// TIA Portal V15.1 export
// export: Created 2019-08-08T13:49:45.9027601Z, ExportSetting None, DisplayName Totally Integrated Automation Portal, DisplayVersion V15.1, DisplayName TIA Portal Openness, DisplayVersion V15.1, DisplayName STEP 7 Professional, DisplayVersion V15.1, DisplayName STEP 7 Safety, DisplayVersion V15.1, DisplayName WinCC Advanced, DisplayVersion V15.1
TYPE "typeSkillStateMachineMapping"
   STRUCT
      StateMachine : Struct
         CurrentState_Id : OPC_UA_NodeId;
         LastTransition_Id : OPC_UA_NodeId;
         AvailableStates_NodeIds : Array[0..2] of OPC_UA_NodeId;
         AvailableStates_Names : Array[0..2] of String;
         AvailableStates_Numbers : Array[0..2] of Byte;
         AvailableTransitions_NodeIds : Array[0..2] of OPC_UA_NodeId;
         AvailableTransitions_Names : Array[0..2] of String;
         AvailableTransitions_Numbers : Array[0..2] of Byte;
      END_STRUCT;
      ClearedStateMachine : Struct
         CurrentState_Id : OPC_UA_NodeId;
         LastTransition_Id : OPC_UA_NodeId;
         AvailableStates_NodeIds : Array[0..3] of OPC_UA_NodeId;
         AvailableStates_Names : Array[0..3] of String;
         AvailableStates_Numbers : Array[0..3] of Byte;
         AvailableTransitions_NodeIds : Array[0..3] of OPC_UA_NodeId;
         AvailableTransitions_Names : Array[0..3] of String;
         AvailableTransitions_Numbers : Array[0..3] of Byte;
      END_STRUCT;
      RunningStateMachine : Struct
         CurrentState_Id : OPC_UA_NodeId;
         LastTransition_Id : OPC_UA_NodeId;
         AvailableStates_NodeIds : Array[0..5] of OPC_UA_NodeId;
         AvailableStates_Names : Array[0..5] of String;
         AvailableStates_Numbers : Array[0..5] of Byte;
         AvailableTransitions_NodeIds : Array[0..6] of OPC_UA_NodeId;
         AvailableTransitions_Names : Array[0..6] of String;
         AvailableTransitions_Numbers : Array[0..6] of Byte;
      END_STRUCT;
      IdleStateMachine : Struct
         CurrentState_Id : OPC_UA_NodeId;
         LastTransition_Id : OPC_UA_NodeId;
         AvailableStates_NodeIds : Array[0..1] of OPC_UA_NodeId;
         AvailableStates_Names : Array[0..1] of String;
         AvailableStates_Numbers : Array[0..1] of Byte;
         AvailableTransitions_NodeIds : Array[0..0] of OPC_UA_NodeId;
         AvailableTransitions_Names : Array[0..0] of String;
         AvailableTransitions_Numbers : Array[0..0] of Byte;
      END_STRUCT;
      HoldStateMachine : Struct
         CurrentState_Id : OPC_UA_NodeId;
         LastTransition_Id : OPC_UA_NodeId;
         AvailableStates_NodeIds : Array[0..2] of OPC_UA_NodeId;
         AvailableStates_Names : Array[0..2] of String;
         AvailableStates_Numbers : Array[0..2] of Byte;
         AvailableTransitions_NodeIds : Array[0..1] of OPC_UA_NodeId;
         AvailableTransitions_Names : Array[0..1] of String;
         AvailableTransitions_Numbers : Array[0..1] of Byte;
      END_STRUCT;
      ResettingStateMachine : Struct
         CurrentState_Id : OPC_UA_NodeId;
         LastTransition_Id : OPC_UA_NodeId;
         AvailableStates_NodeIds : Array[0..2] of OPC_UA_NodeId;
         AvailableStates_Names : Array[0..2] of String;
         AvailableStates_Numbers : Array[0..2] of Byte;
         AvailableTransitions_NodeIds : Array[0..2] of OPC_UA_NodeId;
         AvailableTransitions_Names : Array[0..2] of String;
         AvailableTransitions_Numbers : Array[0..2] of Byte;
      END_STRUCT;
      ExecuteStateMachine : Struct
         CurrentState_Id : OPC_UA_NodeId;
         LastTransition_Id : OPC_UA_NodeId;
         AvailableStates_NodeIds : Array[0..1] of OPC_UA_NodeId;
         AvailableStates_Names : Array[0..1] of String;
         AvailableStates_Numbers : Array[0..1] of Byte;
         AvailableTransitions_NodeIds : Array[0..1] of OPC_UA_NodeId;
         AvailableTransitions_Names : Array[0..1] of String;
         AvailableTransitions_Numbers : Array[0..1] of Byte;
      END_STRUCT;
   END_STRUCT;
   // StateMachine.AvailableStates_NodeIds[0].Identifier := WSTRING#'71';
   // StateMachine.AvailableStates_NodeIds[1].Identifier := WSTRING#'61';
   // StateMachine.AvailableStates_NodeIds[2].Identifier := WSTRING#'62';
   // StateMachine.AvailableStates_Names[0] := 'Cleared';
   // StateMachine.AvailableStates_Names[1] := 'Aborting';
   // StateMachine.AvailableStates_Names[2] := 'Aborted';
   // StateMachine.AvailableStates_Numbers[0] := 1;
   // StateMachine.AvailableStates_Numbers[1] := 2;
   // StateMachine.AvailableStates_Numbers[2] := 3;
   // StateMachine.AvailableTransitions_NodeIds[0].Identifier := WSTRING#'1007';
   // StateMachine.AvailableTransitions_NodeIds[1].Identifier := WSTRING#'1008';
   // StateMachine.AvailableTransitions_NodeIds[2].Identifier := WSTRING#'66';
   // StateMachine.AvailableTransitions_Names[0] := 'ClearedToAborting';
   // StateMachine.AvailableTransitions_Names[1] := 'AbortedToCleared';
   // StateMachine.AvailableTransitions_Names[2] := 'AbortingToAborted';
   // StateMachine.AvailableTransitions_Numbers[0] := 1;
   // StateMachine.AvailableTransitions_Numbers[1] := 2;
   // StateMachine.AvailableTransitions_Numbers[2] := 3;
   // ClearedStateMachine.AvailableStates_NodeIds[0].Identifier := WSTRING#'55';
   // ClearedStateMachine.AvailableStates_NodeIds[1].Identifier := WSTRING#'53';
   // ClearedStateMachine.AvailableStates_NodeIds[2].Identifier := WSTRING#'75';
   // ClearedStateMachine.AvailableStates_NodeIds[3].Identifier := WSTRING#'54';
   // ClearedStateMachine.AvailableStates_Names[0] := 'Clearing';
   // ClearedStateMachine.AvailableStates_Names[1] := 'Stopped';
   // ClearedStateMachine.AvailableStates_Names[2] := 'Running';
   // ClearedStateMachine.AvailableStates_Names[3] := 'Stopping';
   // ClearedStateMachine.AvailableStates_Numbers[0] := 1;
   // ClearedStateMachine.AvailableStates_Numbers[1] := 2;
   // ClearedStateMachine.AvailableStates_Numbers[2] := 3;
   // ClearedStateMachine.AvailableStates_Numbers[3] := 4;
   // ClearedStateMachine.AvailableTransitions_NodeIds[0].Identifier := WSTRING#'58';
   // ClearedStateMachine.AvailableTransitions_NodeIds[1].Identifier := WSTRING#'1000';
   // ClearedStateMachine.AvailableTransitions_NodeIds[2].Identifier := WSTRING#'1006';
   // ClearedStateMachine.AvailableTransitions_NodeIds[3].Identifier := WSTRING#'57';
   // ClearedStateMachine.AvailableTransitions_Names[0] := 'ClearingToStopped';
   // ClearedStateMachine.AvailableTransitions_Names[1] := 'StoppedToRunning';
   // ClearedStateMachine.AvailableTransitions_Names[2] := 'RunningToStopping';
   // ClearedStateMachine.AvailableTransitions_Names[3] := 'StoppingToStopped';
   // ClearedStateMachine.AvailableTransitions_Numbers[0] := 1;
   // ClearedStateMachine.AvailableTransitions_Numbers[1] := 2;
   // ClearedStateMachine.AvailableTransitions_Numbers[2] := 3;
   // ClearedStateMachine.AvailableTransitions_Numbers[3] := 4;
   // RunningStateMachine.AvailableStates_NodeIds[0].Identifier := WSTRING#'27';
   // RunningStateMachine.AvailableStates_NodeIds[1].Identifier := WSTRING#'28';
   // RunningStateMachine.AvailableStates_NodeIds[2].Identifier := WSTRING#'36';
   // RunningStateMachine.AvailableStates_NodeIds[3].Identifier := WSTRING#'1036';
   // RunningStateMachine.AvailableStates_NodeIds[4].Identifier := WSTRING#'37';
   // RunningStateMachine.AvailableStates_NodeIds[5].Identifier := WSTRING#'38';
   // RunningStateMachine.AvailableStates_Names[0] := 'Resetting';
   // RunningStateMachine.AvailableStates_Names[1] := 'Idle';
   // RunningStateMachine.AvailableStates_Names[2] := 'Execute';
   // RunningStateMachine.AvailableStates_Names[3] := 'Hold';
   // RunningStateMachine.AvailableStates_Names[4] := 'Completing';
   // RunningStateMachine.AvailableStates_Names[5] := 'Complete';
   // RunningStateMachine.AvailableStates_Numbers[0] := 1;
   // RunningStateMachine.AvailableStates_Numbers[1] := 2;
   // RunningStateMachine.AvailableStates_Numbers[2] := 3;
   // RunningStateMachine.AvailableStates_Numbers[3] := 4;
   // RunningStateMachine.AvailableStates_Numbers[4] := 5;
   // RunningStateMachine.AvailableStates_Numbers[5] := 6;
   // RunningStateMachine.AvailableTransitions_NodeIds[0].Identifier := WSTRING#'39';
   // RunningStateMachine.AvailableTransitions_NodeIds[1].Identifier := WSTRING#'1002';
   // RunningStateMachine.AvailableTransitions_NodeIds[2].Identifier := WSTRING#'1041';
   // RunningStateMachine.AvailableTransitions_NodeIds[3].Identifier := WSTRING#'1040';
   // RunningStateMachine.AvailableTransitions_NodeIds[4].Identifier := WSTRING#'1003';
   // RunningStateMachine.AvailableTransitions_NodeIds[5].Identifier := WSTRING#'50';
   // RunningStateMachine.AvailableTransitions_NodeIds[6].Identifier := WSTRING#'1042';
   // RunningStateMachine.AvailableTransitions_Names[0] := 'ResettingToIdle';
   // RunningStateMachine.AvailableTransitions_Names[1] := 'IdleToExecute';
   // RunningStateMachine.AvailableTransitions_Names[2] := 'ExecuteToHold';
   // RunningStateMachine.AvailableTransitions_Names[3] := 'HoldToExecute';
   // RunningStateMachine.AvailableTransitions_Names[4] := 'ExecuteToCompleting';
   // RunningStateMachine.AvailableTransitions_Names[5] := 'CompletingToComplete';
   // RunningStateMachine.AvailableTransitions_Names[6] := 'CompleteToIdle';
   // RunningStateMachine.AvailableTransitions_Numbers[0] := 1;
   // RunningStateMachine.AvailableTransitions_Numbers[1] := 2;
   // RunningStateMachine.AvailableTransitions_Numbers[2] := 3;
   // RunningStateMachine.AvailableTransitions_Numbers[3] := 4;
   // RunningStateMachine.AvailableTransitions_Numbers[4] := 5;
   // RunningStateMachine.AvailableTransitions_Numbers[5] := 6;
   // RunningStateMachine.AvailableTransitions_Numbers[6] := 7;
   // IdleStateMachine.AvailableStates_NodeIds[0].Identifier := WSTRING#'1018';
   // IdleStateMachine.AvailableStates_NodeIds[1].Identifier := WSTRING#'1017';
   // IdleStateMachine.AvailableStates_Names[0] := 'InitializeSkill';
   // IdleStateMachine.AvailableStates_Names[1] := 'SkillReady';
   // IdleStateMachine.AvailableStates_Numbers[0] := 1;
   // IdleStateMachine.AvailableStates_Numbers[1] := 2;
   // IdleStateMachine.AvailableTransitions_NodeIds[0].Identifier := WSTRING#'1019';
   // IdleStateMachine.AvailableTransitions_Names[0] := 'InitializeSkillToSkillReady';
   // IdleStateMachine.AvailableTransitions_Numbers[0] := 1;
   // HoldStateMachine.AvailableStates_NodeIds[0].Identifier := WSTRING#'1020';
   // HoldStateMachine.AvailableStates_NodeIds[1].Identifier := WSTRING#'1021';
   // HoldStateMachine.AvailableStates_NodeIds[2].Identifier := WSTRING#'1022';
   // HoldStateMachine.AvailableStates_Names[0] := 'Holding';
   // HoldStateMachine.AvailableStates_Names[1] := 'Held';
   // HoldStateMachine.AvailableStates_Names[2] := 'Unholding';
   // HoldStateMachine.AvailableStates_Numbers[0] := 1;
   // HoldStateMachine.AvailableStates_Numbers[1] := 2;
   // HoldStateMachine.AvailableStates_Numbers[2] := 3;
   // HoldStateMachine.AvailableTransitions_NodeIds[0].Identifier := WSTRING#'1024';
   // HoldStateMachine.AvailableTransitions_NodeIds[1].Identifier := WSTRING#'1023';
   // HoldStateMachine.AvailableTransitions_Names[0] := 'HeldToUnholding';
   // HoldStateMachine.AvailableTransitions_Names[1] := 'HoldingToHeld';
   // HoldStateMachine.AvailableTransitions_Numbers[0] := 1;
   // HoldStateMachine.AvailableTransitions_Numbers[1] := 2;
   // ResettingStateMachine.AvailableStates_NodeIds[0].Identifier := WSTRING#'1026';
   // ResettingStateMachine.AvailableStates_NodeIds[1].Identifier := WSTRING#'1025';
   // ResettingStateMachine.AvailableStates_NodeIds[2].Identifier := WSTRING#'1027';
   // ResettingStateMachine.AvailableStates_Names[0] := 'CheckSkillComponent';
   // ResettingStateMachine.AvailableStates_Names[1] := 'InitializeSkillComponent';
   // ResettingStateMachine.AvailableStates_Names[2] := 'SkillComponentsReady';
   // ResettingStateMachine.AvailableStates_Numbers[0] := 1;
   // ResettingStateMachine.AvailableStates_Numbers[1] := 2;
   // ResettingStateMachine.AvailableStates_Numbers[2] := 3;
   // ResettingStateMachine.AvailableTransitions_NodeIds[0].Identifier := WSTRING#'1028';
   // ResettingStateMachine.AvailableTransitions_NodeIds[1].Identifier := WSTRING#'10230';
   // ResettingStateMachine.AvailableTransitions_NodeIds[2].Identifier := WSTRING#'1029';
   // ResettingStateMachine.AvailableTransitions_Names[0] := 'CheckSkillComponentToInitializeSkillComponent';
   // ResettingStateMachine.AvailableTransitions_Names[1] := 'CheckSkillComponentToSkillComponentsReady';
   // ResettingStateMachine.AvailableTransitions_Names[2] := 'InitializeSkillComponentToCheckSkillComponent';
   // ResettingStateMachine.AvailableTransitions_Numbers[0] := 1;
   // ResettingStateMachine.AvailableTransitions_Numbers[1] := 2;
   // ResettingStateMachine.AvailableTransitions_Numbers[2] := 3;
   // ExecuteStateMachine.AvailableStates_NodeIds[0].Identifier := WSTRING#'1013';
   // ExecuteStateMachine.AvailableStates_NodeIds[1].Identifier := WSTRING#'1014';
   // ExecuteStateMachine.AvailableStates_Names[0] := 'ExecuteSkill';
   // ExecuteStateMachine.AvailableStates_Names[1] := 'WaitForNextStep';
   // ExecuteStateMachine.AvailableStates_Numbers[0] := 1;
   // ExecuteStateMachine.AvailableStates_Numbers[1] := 2;
   // ExecuteStateMachine.AvailableTransitions_NodeIds[0].Identifier := WSTRING#'1015';
   // ExecuteStateMachine.AvailableTransitions_NodeIds[1].Identifier := WSTRING#'1016';
   // ExecuteStateMachine.AvailableTransitions_Names[0] := 'ExecuteSkillToWaitForNextStep';
   // ExecuteStateMachine.AvailableTransitions_Names[1] := 'WaitForNextStepToExecuteSkill';
   // ExecuteStateMachine.AvailableTransitions_Numbers[0] := 1;
   // ExecuteStateMachine.AvailableTransitions_Numbers[1] := 2;
END_TYPE
